PROGRAM MAIN
VAR
	bPageUp : BOOL;
	bPageDown : BOOL;
END_VAR

END_PROGRAM

(* stored: Version 1.1.0.1
   POU MAIN: Id {00c02a50-f51b-4ee4-a927-7ab9b30d1799}, SpecialFunc None *)
